VAR_GLOBAL // INPUTS
    ivar_M_p_i AT %I*: LREAL;
END_VAR

(* stored: ProductVersion 3.1.0.18, Version 1.1.0.1 *)
